(* CoDeSys 2.3 export: STRMODBUSUZSTATUS.EXP *)

(* Data type *)
TYPE strModbusUZStatus :
STRUCT
	Ready : BOOL;
	Running : BOOL;
	Fail	: BOOL;
	Signal : tUZSignal;
END_STRUCT
END_TYPE
